// TIA Portal project "ISA_P7" (V16)

(* hardware
DEVICE "S7-1200 station_1"  S7-1200 Station
   slot 0: "Rack_0"  S7-1200 Rack  Rack  V1.0
   slot 1: "PLC_1"  CPU 1215C DC/DC/DC  6ES7 215-1AG40-0XB0  V4.4
DEVICE "SINAMICS G_1"  Sinamics.Device
   slot 0: "	_0"  Rail  SinamicsG120SVecto
   slot 0: "Accionamiento_1"  G120 CU250S-2 PN Vector  6SL3246-0BA22-1FA0  4.7.10
      slot 1: "Interfaz PROFINET"  MDD-SinamicsG120-P
   slot 3: "PM240 IP20"  PM240 IP20  6SL3224-0BE13-7UA0  -
DEVICE "PC-System_1"  SIMATIC PC station
   slot 0: "Estación PC SIMATIC"  Rail  SIMATIC PC-Station  V1.0
      slot 125: "Stationmanager"  Station_Manager  V6.0.4
   slot 1: "HMI_RT_1"  WinCC RT Advanced  6AV2 104-0xxxx-xxxx  16.0.0.0
      slot 33792: "Interfaz del equipo"  Host interface
   slot 2: "IE general_1"  IE General  IE_CP  V8.2.0
*)

// ===== PLC "PLC_1"  CPU 1215C DC/DC/DC =====

VAR_GLOBAL   // PLC tag table "Tabla de variables estándar"
   "ConexiónMotor" AT %Q0.0 : Bool;
   "InversionSentido" AT %Q0.3 : Bool;
   "ConsignaVelocidad" AT %QW64 : Int;
   "ConsignaVelocidadAlcanzada" AT %I0.0 : Bool;
   "ActivarJog1" AT %Q0.2 : Bool;
   "VelocidadActual" AT %IW64 : Word;
   "FinalCarrera" AT %I0.4 : Bool;
   "Etapa0" AT %M10.0 : Bool;
   "Etapa1" AT %M10.1 : Bool;
   "Etapa2" AT %M10.2 : Bool;
   "Etapa3" AT %M10.3 : Bool;
   "Etapa4" AT %M10.4 : Bool;
   "Etapa5" AT %M10.5 : Bool;
   "Etapa6" AT %M10.6 : Bool;
   "Etapa7" AT %M10.7 : Bool;
   "System_Byte" AT %MB1 : Byte;
   "FirstScan" AT %M1.0 : Bool;
   "DiagStatusUpdate" AT %M1.1 : Bool;
   "AlwaysTRUE" AT %M1.2 : Bool;
   "AlwaysFALSE" AT %M1.3 : Bool;
   "BitInterrupción" AT %M100.0 : Bool;
   "Tag_1" AT %M90.0 : Bool;
   "Etapas0-7" AT %MB10 : Byte;
   "Clock_Byte" AT %MB0 : Byte;
   "Clock_10Hz" AT %M0.0 : Bool;
   "Clock_5Hz" AT %M0.1 : Bool;
   "Clock_2.5Hz" AT %M0.2 : Bool;
   "Clock_2Hz" AT %M0.3 : Bool;
   "Clock_1.25Hz" AT %M0.4 : Bool;
   "Clock_1Hz" AT %M0.5 : Bool;
   "Clock_0.625Hz" AT %M0.6 : Bool;
   "Clock_0.5Hz" AT %M0.7 : Bool;
END_VAR

DATA_BLOCK "Variables"   // DB1
{ S7_Optimized_Access := 'TRUE' }
VERSION : 0.1
   VAR
      ConexionMotorScada : Bool;
      AutomaticoScada : Bool;
      MarchaScada : Bool;
      ConsignaAlcanzadaScada : Bool;
      InversionMotorScada : Bool;
      VelocidadActualScada : Bool;
      ActivarJog1Scada : Bool;
      VelocidadMotorScada : Int;
      VelocidadNormalizada : Real;
      VelocidadEscalada : Int;
      VelocidadReal : Real;
      Posiciones : Array[0..4] of Int;
      PosicionesMilimetrosScada : Array[0..4] of Int;
      Puntero : SInt;
      Posicion : SInt;
      ResolucionEncoderScada : DInt;
      PosicionProximaAbajo : DInt;
      PosicionProximaArriba : DInt;
      EntradaFinalizada : Bool;
      CambioVelocidadScada : DInt;
   END_VAR
   VAR RETAIN
      PulsosEncoder : Int;
   END_VAR
BEGIN
   Posiciones[0] := 3000;
   Posiciones[1] := 6000;
   Posiciones[2] := 9000;
   Posiciones[3] := 12000;
   Posiciones[4] := 15000;
END_DATA_BLOCK

DATA_BLOCK "VelocidadReal"   // DB2
{ S7_Optimized_Access := 'TRUE' }
VERSION : 0.1
// stored: InstanceOfName Analog_IN
"Analog_IN"
BEGIN
END_DATA_BLOCK

DATA_BLOCK "Calculo_milimetros_DB"   // DB4
{ S7_Optimized_Access := 'TRUE' }
VERSION : 0.1
// stored: InstanceOfName Calculo_milimetros
"Calculo_milimetros"
BEGIN
END_DATA_BLOCK

DATA_BLOCK "Analog_OUT_DB"   // DB5
{ S7_Optimized_Access := 'TRUE' }
VERSION : 0.1
// stored: InstanceOfName Analog_OUT
"Analog_OUT"
BEGIN
END_DATA_BLOCK

DATA_BLOCK "Encoder_Control"   // DB7
{ S7_Optimized_Access := 'TRUE' }
VERSION : 0.1
   VAR
      MyHSC : HSC_Count;
   END_VAR
BEGIN
   MyHSC.EnReference1 := 1;
   MyHSC.EnSync := 1;
   MyHSC.EnHSC := 1;
END_DATA_BLOCK

// folder: System blocks/Program resources

DATA_BLOCK "Timer1"   // DB3
{ S7_Optimized_Access := 'TRUE' }
AUTHOR : Simatic
FAMILY : IEC
NAME : IEC_TMR
VERSION : 1.0
// stored: InstanceOfName IEC_TIMER
"IEC_TIMER"
BEGIN
END_DATA_BLOCK

DATA_BLOCK "ton"   // DB8
{ S7_Optimized_Access := 'TRUE' }
AUTHOR : Simatic
FAMILY : IEC
NAME : IEC_TMR
VERSION : 1.0
// stored: InstanceOfName IEC_TIMER
"IEC_TIMER"
BEGIN
   PT := T#500MS;
END_DATA_BLOCK

// folder: (top level)

FUNCTION_BLOCK "Calculo_milimetros"   // FB1, SCL
{ S7_Optimized_Access := 'TRUE' }
VERSION : 0.1
   VAR_INPUT
      Lectura_pulsos : DInt;
      Radio : Real;
      Resolucion_encoder : Int;
   END_VAR
   VAR_OUTPUT
      mm_recorridos : Real;
   END_VAR
   VAR CONSTANT
      pi : Real := 3.1415;
   END_VAR
BEGIN
   #mm_recorridos := (#Lectura_pulsos * #Radio * 2 * #pi) / #Resolucion_encoder;
END_FUNCTION_BLOCK

FUNCTION_BLOCK "Analog_IN"   // FB4, LAD
{ S7_Optimized_Access := 'TRUE' }
VERSION : 0.1
   VAR_INPUT
      Input : Int;
      X_min : Real;
      X_max : Real;
      Y_min : Real;
      Y_max : Real;
      IsTension : Bool;
   END_VAR
   VAR_OUTPUT
      Output : Real;
   END_VAR
   VAR
      X_min_bits : Int;
      X_max_bits : Int;
      norm : Real;
   END_VAR
   VAR CONSTANT
      tension_pendent : Real := 2764.8;
      intensity_pendent : Real := 1382.4;
   END_VAR
BEGIN

REGION Network 1 (SCL)

   IF #IsTension THEN
       #X_min_bits := REAL_TO_INT(#X_min * #tension_pendent);
       #X_max_bits := REAL_TO_INT(#X_max * #tension_pendent);
   ELSE
       #X_min_bits := REAL_TO_INT(#X_min * #intensity_pendent);
       #X_max_bits := REAL_TO_INT(#X_max * #intensity_pendent);
   END_IF;
END_REGION

REGION Network 2
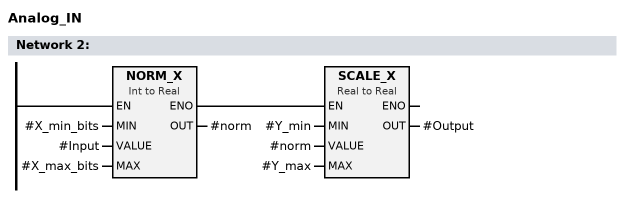
   RUNG wire#powerrail
      { S7_Templates := "[SrcType := Int, DestType := Real]" } Normalize(min := #X_min_bits, value := #Input, max := #X_max_bits, out => #norm)
      { S7_Templates := "[SrcType := Real, DestType := Real]" } Scale(min := #Y_min, value := #norm, max := #Y_max, out => #Output)
   END_RUNG
   // the same network as SCL:
   #norm := NORM_X(MIN := #X_min_bits, VALUE := #Input, MAX := #X_max_bits);
   #Output := SCALE_X(MIN := #Y_min, VALUE := #norm, MAX := #Y_max);
END_REGION
END_FUNCTION_BLOCK

FUNCTION_BLOCK "Analog_OUT"   // FB5, LAD
{ S7_Optimized_Access := 'TRUE' }
VERSION : 0.1
   VAR_INPUT
      Input : Real;
      X_min : Real;
      X_max : Real;
      Y_min : Real;
      Y_max : Real;
      IsTension : Bool;
   END_VAR
   VAR_OUTPUT
      Output : Int;
   END_VAR
   VAR
      Y_min_bits : Int;
      Y_max_bits : Int;
      norm : Real;
   END_VAR
   VAR CONSTANT
      tension_pendent : Real := 2764.8;
      intensity_pendent : Real := 1382.4;
   END_VAR
BEGIN

REGION Network 1 (SCL)

   IF #IsTension THEN
       #Y_min_bits := REAL_TO_INT(#Y_min * #tension_pendent);
       #Y_max_bits := REAL_TO_INT(#Y_max * #tension_pendent);
   ELSE
       #Y_min_bits := REAL_TO_INT(#Y_min * #intensity_pendent);
       #Y_max_bits := REAL_TO_INT(#Y_max * #intensity_pendent);
   END_IF;
END_REGION

REGION Network 2
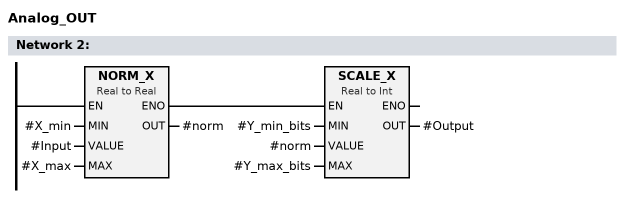
   RUNG wire#powerrail
      { S7_Templates := "[SrcType := Real, DestType := Real]" } Normalize(min := #X_min, value := #Input, max := #X_max, out => #norm)
      { S7_Templates := "[SrcType := Real, DestType := Int]" } Scale(min := #Y_min_bits, value := #norm, max := #Y_max_bits, out => #Output)
   END_RUNG
   // the same network as SCL:
   #norm := NORM_X(MIN := #X_min, VALUE := #Input, MAX := #X_max);
   #Output := SCALE_X(MIN := #Y_min_bits, VALUE := #norm, MAX := #Y_max_bits);
END_REGION
END_FUNCTION_BLOCK

ORGANIZATION_BLOCK "Variador"   // OB1, LAD, ProgramCycle
TITLE = "Main Program Sweep (Cycle)"
{ S7_Optimized_Access := 'TRUE' }
VERSION : 0.1
   VAR_INPUT
      Initial_Call : Bool;   // Initial call of this OB
      Remanence : Bool;   // =True, if remanent data are available
   END_VAR
BEGIN

REGION Network 1: Escalado consigna de velocidad
   // Varia la consigna de velocidad que recibe el variador (señal de 0 a 20mA) en función del deslizante en SCADA (señal de 0 a 1800).
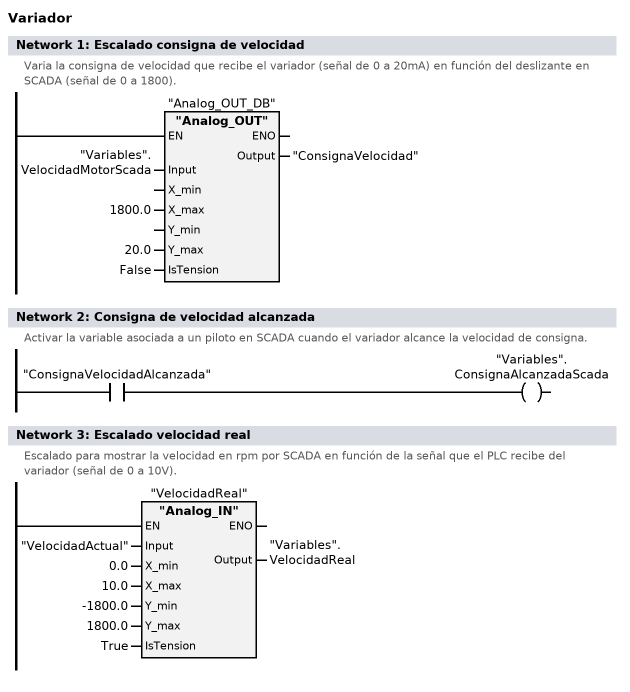
   RUNG wire#powerrail
      "Analog_OUT_DB"(Input := "Variables".VelocidadMotorScada, X_min :=, X_max := 1800.0, Y_min :=, Y_max := 20.0, IsTension := False, Output => "ConsignaVelocidad")
   END_RUNG
   // the same network as SCL:
   "Analog_OUT_DB"(Input := "Variables".VelocidadMotorScada,   // "Analog_OUT"
                   X_max := 1800.0,
                   Y_max := 20.0,
                   IsTension := False,
                   Output => "ConsignaVelocidad");
END_REGION

REGION Network 2: Consigna de velocidad alcanzada
   // Activar la variable asociada a un piloto en SCADA cuando el variador alcance la velocidad de consigna.
   RUNG wire#powerrail
      Contact( "ConsignaVelocidadAlcanzada" )
      Coil( "Variables".ConsignaAlcanzadaScada )
   END_RUNG
   // the same network as SCL:
   "Variables".ConsignaAlcanzadaScada := "ConsignaVelocidadAlcanzada";
END_REGION

REGION Network 3: Escalado velocidad real
   // Escalado para mostrar la velocidad en rpm por SCADA en función de la señal que el PLC recibe del variador (señal de 0 a 10V).
   RUNG wire#powerrail
      "VelocidadReal"(Input := "VelocidadActual", X_min := 0.0, X_max := 10.0, Y_min := -1800.0, Y_max := 1800.0, IsTension := True, Output => "Variables".VelocidadReal)
   END_RUNG
   // the same network as SCL:
   "VelocidadReal"(Input := "VelocidadActual",   // "Analog_IN"
                   X_min := 0.0,
                   X_max := 10.0,
                   Y_min := -1800.0,
                   Y_max := 1800.0,
                   IsTension := True,
                   Output => "Variables".VelocidadReal);
END_REGION
END_ORGANIZATION_BLOCK

ORGANIZATION_BLOCK "Interrupción"   // OB40, SCL, HWProcessInterrupt
{ S7_Optimized_Access := 'TRUE' }
VERSION : 0.1
   VAR_INPUT
      LADDR : Hw_Io;   // Hardware identifier
      USI : Word;   // User structure identifier
      IChannel : USInt;   // Interrupt channel number
      EventType : Byte;   // EventType
   END_VAR
BEGIN
   "Variables".Puntero += 1;
   "BitInterrupción" := 1;
END_ORGANIZATION_BLOCK

ORGANIZATION_BLOCK "Encoder"   // OB123, LAD, ProgramCycle
TITLE = "Main Program Sweep (Cycle)"
{ S7_Optimized_Access := 'TRUE' }
VERSION : 0.1
   VAR_INPUT
      Initial_Call : Bool;   // Initial call of this OB
      Remanence : Bool;   // =True, if remanent data are available
   END_VAR
BEGIN

REGION Network 1: Control del encoder
   // Asociar el encoder al bloque de control.
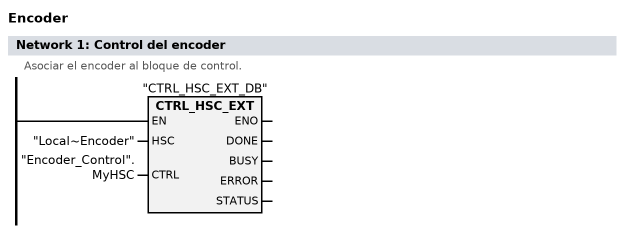
   "CTRL_HSC_EXT_DB"(HSC := "Local~Encoder", CTRL := "Encoder_Control".MyHSC);   // CTRL_HSC_EXT
END_REGION

REGION Network 2 (SCL): Constantes del control del encoder
   // Activar el bit de contaje para registrar los pulsos del encoder.
   "Encoder_Control".MyHSC.EnHSC := 1;
   // Activar el bit de puerta de sincronización para reiniciar el encoder de forma externa.
   "Encoder_Control".MyHSC.EnSync := 1;
   // Activar la referencia 1 para generar una interrupción cuando se alcance dicha referencia.
   "Encoder_Control".MyHSC.EnReference1 := 1;
END_REGION
END_ORGANIZATION_BLOCK

ORGANIZATION_BLOCK "Grafcet Principal"   // OB124, LAD, ProgramCycle
TITLE = "Main Program Sweep (Cycle)"
{ S7_Optimized_Access := 'TRUE' }
VERSION : 0.1
   VAR_INPUT
      Initial_Call : Bool;   // Initial call of this OB
      Remanence : Bool;   // =True, if remanent data are available
   END_VAR
BEGIN

REGION Network 1
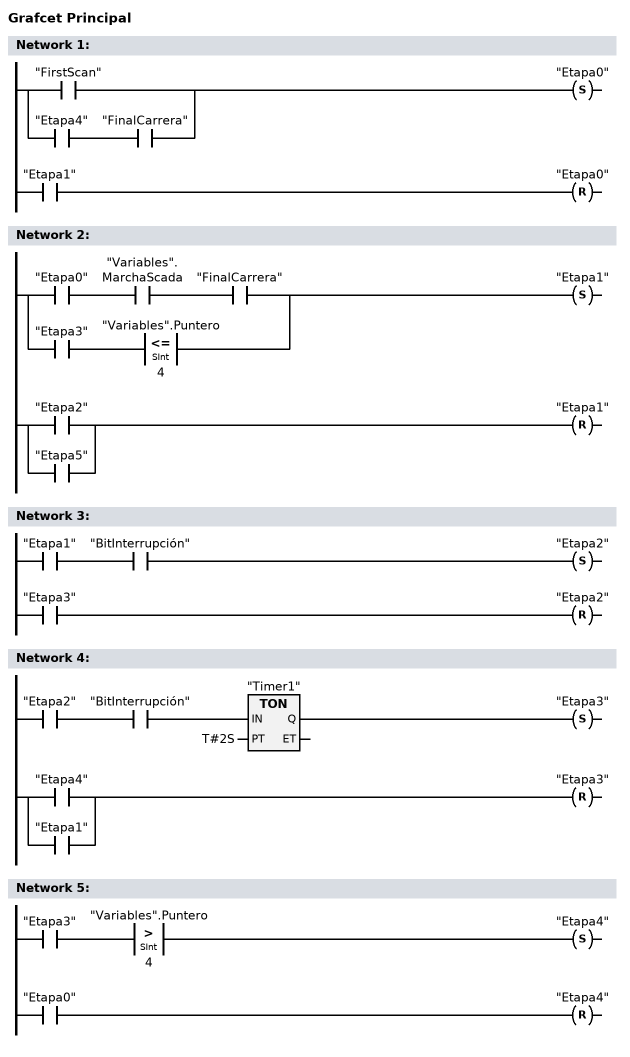
   RUNG wire#powerrail
      Contact( "FirstScan" )
      wire#w1
      S_Coil( "Etapa0" )
   END_RUNG
   RUNG wire#powerrail
      Contact( "Etapa4" )
      Contact( "FinalCarrera" )
   END_RUNG wire#w1
   RUNG wire#powerrail
      Contact( "Etapa1" )
      R_Coil( "Etapa0" )
   END_RUNG
   // the same network as SCL:
   IF "FirstScan" OR ("Etapa4" AND "FinalCarrera") THEN "Etapa0" := TRUE; END_IF;
   IF "Etapa1" THEN "Etapa0" := FALSE; END_IF;
END_REGION

REGION Network 2
   RUNG wire#powerrail
      Contact( "Etapa0" )
      Contact( "Variables".MarchaScada )
      Contact( "FinalCarrera" )
      wire#w1
      S_Coil( "Etapa1" )
   END_RUNG
   RUNG wire#powerrail
      Contact( "Etapa3" )
      { S7_Templates := "SrcType := SInt" } LE_Contact(in1 := "Variables".Puntero, in2 := 4)
   END_RUNG wire#w1
   RUNG wire#powerrail
      Contact( "Etapa2" )
      wire#w2
      R_Coil( "Etapa1" )
   END_RUNG
   RUNG wire#powerrail
      Contact( "Etapa5" )
   END_RUNG wire#w2
   // the same network as SCL:
   IF ("Etapa0" AND "Variables".MarchaScada AND "FinalCarrera") OR ("Etapa3" AND ("Variables".Puntero <= 4)) THEN
       "Etapa1" := TRUE;
   END_IF;
   IF "Etapa2" OR "Etapa5" THEN "Etapa1" := FALSE; END_IF;
END_REGION

REGION Network 3
   RUNG wire#powerrail
      Contact( "Etapa1" )
      Contact( "BitInterrupción" )
      S_Coil( "Etapa2" )
   END_RUNG
   RUNG wire#powerrail
      Contact( "Etapa3" )
      R_Coil( "Etapa2" )
   END_RUNG
   // the same network as SCL:
   IF "Etapa1" AND "BitInterrupción" THEN "Etapa2" := TRUE; END_IF;
   IF "Etapa3" THEN "Etapa2" := FALSE; END_IF;
END_REGION

REGION Network 4
   "Timer1".TON(IN := "Etapa2" AND "BitInterrupción", PT := T#2S);
   IF "Timer1".Q THEN "Etapa3" := TRUE; END_IF;
   IF "Etapa4" OR "Etapa1" THEN "Etapa3" := FALSE; END_IF;
END_REGION

REGION Network 5
   RUNG wire#powerrail
      Contact( "Etapa3" )
      { S7_Templates := "SrcType := SInt" } GT_Contact(in1 := "Variables".Puntero, in2 := 4)
      S_Coil( "Etapa4" )
   END_RUNG
   RUNG wire#powerrail
      Contact( "Etapa0" )
      R_Coil( "Etapa4" )
   END_RUNG
   // the same network as SCL:
   IF "Etapa3" AND ("Variables".Puntero > 4) THEN "Etapa4" := TRUE; END_IF;
   IF "Etapa0" THEN "Etapa4" := FALSE; END_IF;
END_REGION

REGION Network 6 (SCL)
   IF NOT "Variables".AutomaticoScada THEN
       "Etapas0-7" := 2#00000001;
   END_IF;
END_REGION
END_ORGANIZATION_BLOCK

ORGANIZATION_BLOCK "Salidas"   // OB125, LAD, ProgramCycle
TITLE = "Main Program Sweep (Cycle)"
{ S7_Optimized_Access := 'TRUE' }
VERSION : 0.1
   VAR_INPUT
      Initial_Call : Bool;   // Initial call of this OB
      Remanence : Bool;   // =True, if remanent data are available
   END_VAR
BEGIN

REGION Network 1
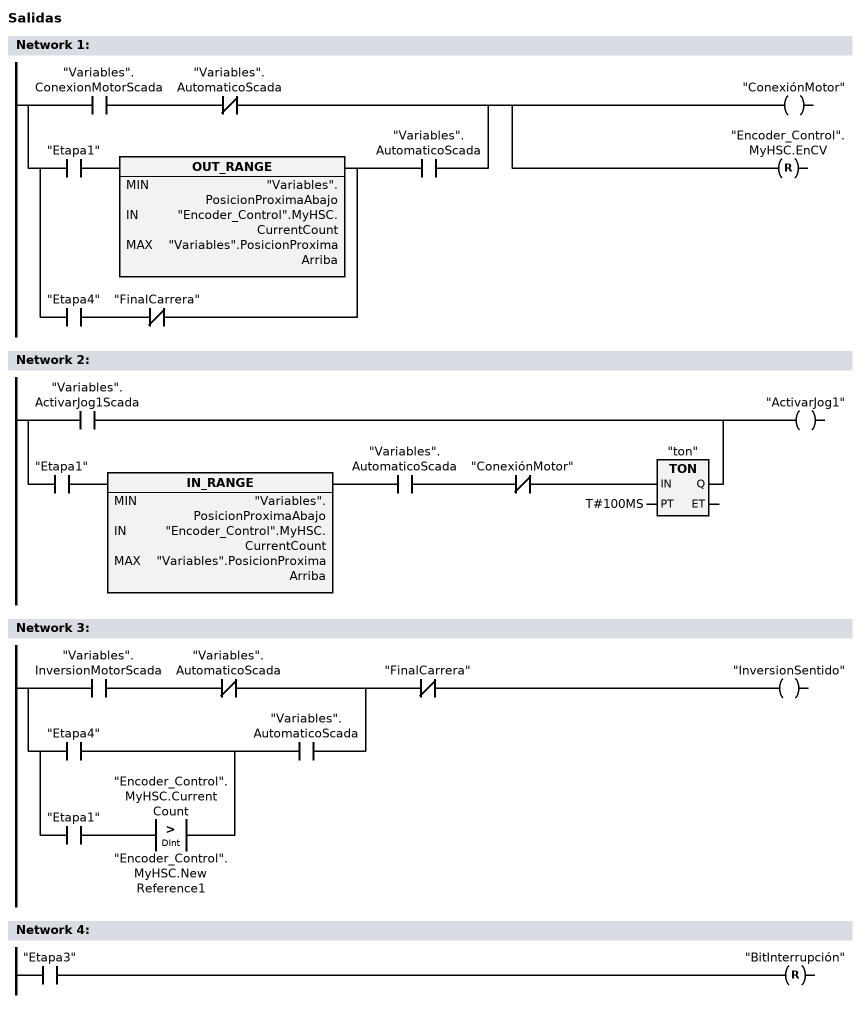
   "ConexiónMotor" := ("Variables".ConexionMotorScada AND NOT "Variables".AutomaticoScada) OR ((("Etapa1" AND (("Encoder_Control".MyHSC.CurrentCount < "Variables".PosicionProximaAbajo) OR ("Encoder_Control".MyHSC.CurrentCount > "Variables".PosicionProximaArriba))) OR ("Etapa4" AND NOT "FinalCarrera")) AND "Variables".AutomaticoScada);
   IF "ConexiónMotor" THEN "Encoder_Control".MyHSC.EnCV := FALSE; END_IF;
END_REGION

REGION Network 2
   "ton".TON(IN := "Etapa1" AND ("Variables".PosicionProximaAbajo <= "Encoder_Control".MyHSC.CurrentCount) AND ("Encoder_Control".MyHSC.CurrentCount <= "Variables".PosicionProximaArriba) AND "Variables".AutomaticoScada AND NOT "ConexiónMotor",
             PT := T#100MS);
   "ActivarJog1" := "Variables".ActivarJog1Scada OR "ton".Q;
END_REGION

REGION Network 3
   RUNG wire#powerrail
      Contact( "Variables".InversionMotorScada )
      I_Contact( "Variables".AutomaticoScada )
      wire#w1
      I_Contact( "FinalCarrera" )
      Coil( "InversionSentido" )
   END_RUNG
   RUNG wire#powerrail
      Contact( "Etapa4" )
      wire#w2
      Contact( "Variables".AutomaticoScada )
   END_RUNG wire#w1
   RUNG wire#powerrail
      Contact( "Etapa1" )
      { S7_Templates := "SrcType := DInt" } GT_Contact(in1 := "Encoder_Control".MyHSC.CurrentCount, in2 := "Encoder_Control".MyHSC.NewReference1)
   END_RUNG wire#w2
   // the same network as SCL:
   "InversionSentido" := (("Variables".InversionMotorScada AND NOT "Variables".AutomaticoScada) OR (("Etapa4" OR ("Etapa1" AND ("Encoder_Control".MyHSC.CurrentCount > "Encoder_Control".MyHSC.NewReference1))) AND "Variables".AutomaticoScada)) AND NOT "FinalCarrera";
END_REGION

REGION Network 4
   RUNG wire#powerrail
      Contact( "Etapa3" )
      R_Coil( "BitInterrupción" )
   END_RUNG
   // the same network as SCL:
   IF "Etapa3" THEN "BitInterrupción" := FALSE; END_IF;
END_REGION
END_ORGANIZATION_BLOCK

ORGANIZATION_BLOCK "Posición"   // OB126, SCL, ProgramCycle
TITLE = "Main Program Sweep (Cycle)"
{ S7_Optimized_Access := 'TRUE' }
VERSION : 0.1
   VAR_INPUT
      Initial_Call : Bool;   // Initial call of this OB
      Remanence : Bool;   // =True, if remanent data are available
   END_VAR
BEGIN
   IF "FirstScan" THEN
       "Encoder_Control".MyHSC.NewReference1 := "Variables".Posiciones[0];
       "Variables".Puntero := 0;
       "Encoder_Control".MyHSC.NewCurrentCount := "Variables".PulsosEncoder;
       "Encoder_Control".MyHSC.EnCV := 1;
   END_IF;

   "Variables".PulsosEncoder := "Encoder_Control".MyHSC.CurrentCount;

   IF "BitInterrupción" THEN
       IF "Etapa0" THEN
           "Variables".Puntero := 0;
       END_IF;
       "Encoder_Control".MyHSC.NewReference1 := "Variables".Posiciones["Variables".Puntero];
   END_IF;

   IF "Variables".EntradaFinalizada THEN
       FOR "Variables".Posicion := 0 TO 4 DO
           "Variables".Posiciones["Variables".Posicion] := ("Variables".PosicionesMilimetrosScada["Variables".Posicion] * "Variables".ResolucionEncoderScada) / 5;
       END_FOR;
       "Variables".EntradaFinalizada := 0;
   END_IF;

   "Variables".PosicionProximaAbajo := "Encoder_Control".MyHSC.NewReference1 * "Variables".CambioVelocidadScada / 100;
   "Variables".PosicionProximaArriba := "Encoder_Control".MyHSC.NewReference1 * (200 - "Variables".CambioVelocidadScada) / 100;
END_ORGANIZATION_BLOCK

(* ===== HMI "HMI_RT_1" =====
system functions are stored by id; their names below are inferred from use
connection "HMI_Conexión_1": ETHERNET, S7_1200_OMS

HMI tags "Tabla de variables estándar"
   "Variables_AvanceMotorScada" : Bool = PLC Variables.ConexionMotorScada, 1 s
   "Variables_RetrocesoMotorScada" : Bool = PLC Variables.InversionMotorScada, 1 s
   "Variables_VelocidadMotorScada" : Int = PLC Variables.VelocidadMotorScada, 1 s
   "Variables_VelocidadConsignaAlcanzada" : Bool = PLC Variables.ConsignaAlcanzadaScada, 1 s
   "Variables_ActivarJog1Scada" : Bool = PLC Variables.ActivarJog1Scada, 1 s
   "Variables_VelocidadReal" : Real = PLC Variables.VelocidadReal, 1 s
   "Variables_VelocidadEscalada" : Int = PLC Variables.VelocidadEscalada, 1 s
   "Variables_MarchaScada" : Bool = PLC Variables.MarchaScada, 1 s
   "Variables_Posiciones{0}" : Int = PLC Variables.Posiciones[0], 1 s
   "Variables_Posiciones{4}" : Int = PLC Variables.Posiciones[4], 1 s
   "Variables_AutomaticoScada" : Bool = PLC Variables.AutomaticoScada, 1 s
   "Variables_PosicionesMilimetrosScada{0}" : Int = PLC Variables.PosicionesMilimetrosScada[0], 1 s
   "Variables_PosicionesMilimetrosScada{1}" : Int = PLC Variables.PosicionesMilimetrosScada[1], 1 s
   "Variables_PosicionesMilimetrosScada{2}" : Int = PLC Variables.PosicionesMilimetrosScada[2], 1 s
   "Variables_PosicionesMilimetrosScada{3}" : Int = PLC Variables.PosicionesMilimetrosScada[3], 1 s
   "Variables_PosicionesMilimetrosScada{4}" : Int = PLC Variables.PosicionesMilimetrosScada[4], 1 s
   "Variables_EntradaFinalizada" : Bool = PLC Variables.EntradaFinalizada, 1 s
   "Variables_ResolucionEncoderScada" : DInt = PLC Variables.ResolucionEncoderScada, 1 s
   "Variables_CambioVelocidadScada" : DInt = PLC Variables.CambioVelocidadScada, 1 s

screen "Imagen_1" 800x600
   Button "Botón_1" at 63,57 size 96x32; TextOff 'Conexión'
      on Click: InvertBit("Variables_AvanceMotorScada")
   TextField "Campo de texto_1" at 299,79 size 135x47; Text 'Velocidad'
   Slider "Deslizador_1" at 299,126 size 80x449; Caption 'SIMATIC'
      ProcessValue <- "Variables_VelocidadMotorScada"
   Circle "Círculo_1" at 91,387 size 48x48
      Appearance <- "Variables_VelocidadConsignaAlcanzada"
   TextField "Campo de texto_2" at 4,329 size 214x55; Text 'Velocidad Consigna Alcanzada'
   TextField "Campo de texto_3" at 22,22 size 198x22; Text 'Movimiento Manual'
   Button "Botón_3" at 78,279 size 74x32; TextOff 'JOG1'
      on Press: SetBit("Variables_ActivarJog1Scada")
      on Release: ResetBit("Variables_ActivarJog1Scada")
   TextField "Campo de texto_4" at 9,208 size 201x57; Text 'Activar JOG1 v = 400rpm'
   IOField "Campo ES_1" at 50,495 size 131x32; FormatPattern s9999.99; Unit rpm
      ProcessValue <- "Variables_VelocidadReal"
   TextField "Campo de texto_5" at 51,458 size 263x22; Text 'Velocidad Actual'
   Switch "Interruptor_1" at 56,109 size 120x88; CaptionText 'Inversión'; TextOff 'OFF'; TextOn 'ON'
      ProcessValue <- "Variables_RetrocesoMotorScada"
   Button "Botón_2" at 521,159 size 96x32; TextOff 'Marcha'
      on Press: SetBit("Variables_MarchaScada")
      on Release: ResetBit("Variables_MarchaScada")
   TextField "Campo de texto_6" at 478,124 size 198x22; Text 'Movimiento Automático'
   TextField "Campo de texto_7" at 533,205 size 198x22; Text 'Posiciones (mm)'
   IOField "Campo ES_2" at 547,246 size 53x32; FormatPattern 999
      ProcessValue <- "Variables_PosicionesMilimetrosScada{0}"
   TextField "Campo de texto_8" at 441,249 size 102x22; Text 'Posición 1'
   IOField "Campo ES_3" at 547,300 size 53x32; FormatPattern 999
      ProcessValue <- "Variables_PosicionesMilimetrosScada{1}"
   TextField "Campo de texto_9" at 441,303 size 101x22; Text 'Posición 2'
   IOField "Campo ES_4" at 547,356 size 53x32; FormatPattern 999
      ProcessValue <- "Variables_PosicionesMilimetrosScada{2}"
   TextField "Campo de texto_10" at 441,359 size 98x22; Text 'Posición 3'
   IOField "Campo ES_5" at 716,246 size 53x32; FormatPattern 999
      ProcessValue <- "Variables_PosicionesMilimetrosScada{3}"
   TextField "Campo de texto_11" at 610,249 size 99x22; Text 'Posición 4'
   IOField "Campo ES_6" at 716,301 size 53x32; FormatPattern 999
      ProcessValue <- "Variables_PosicionesMilimetrosScada{4}"
   TextField "Campo de texto_12" at 610,304 size 100x22; Text 'Posición 5'
   Switch "Interruptor_2" at 280,21 size 120x58; TextOn 'ON'; CaptionText 'Automático'; TextOff 'OFF'
      ProcessValue <- "Variables_AutomaticoScada"
   IOField "Campo ES_7" at 628,43 size 52x32; FormatPattern 999
      ProcessValue <- "Variables_ResolucionEncoderScada"
   TextField "Campo de texto_13" at 459,46 size 153x22; Text 'Resolución Encoder'
   Button "Botón_4" at 640,356 size 96x32; TextOff 'Guardar'
      on Release: ResetBit("Variables_EntradaFinalizada")
      on Press: SetBit("Variables_EntradaFinalizada")
   IOField "Campo ES_8" at 707,410 size 53x32; FormatPattern 999
      ProcessValue <- "Variables_CambioVelocidadScada"
   TextField "Campo de texto_14" at 458,413 size 241x22; Text 'Cambio a velocidad lenta (%)'
*)